Fanuc KAREL source: kb00043.KL

PROGRAM KB00043
%STACKSIZE=65535
%PRIORITY=65535
%NOLOCKGROUP
VAR
P1 : INTEGER
P2 : STRING[80]
BEGIN
P1=1
P2='A'
CNV_TIME_STR(P1,P2)
END KB00043
